{attribute 'pack_mode' := '1'}
TYPE ChangeOutputLine EXTENDS IncomingMessage :
STRUCT
	lineIndex: DINT;
	newState: BOOL;
END_STRUCT
END_TYPE

(* stored: Version 1.1.0.1, ProductVersion 3.1.4022.12
   DUT ChangeOutputLine: Id {f6361086-b9f6-4a55-9af2-baf4425345d4} *)
